# EPICS substitutions: EMIL_PZI_00App/Db/user.substitutions
# Example substitutions file

file "db/circle.db" {
    { user = "emil" }
}

file "db/dbExample1.db" {
    { user = "emil" }
}

file db/dbExample2.db {
    pattern { user, no, scan }
        { "emil", 1, "1 second" }
        { "emil", 2, "2 second" }
        { "emil", 3, "5 second" }
}
